FUNCTION ASSEMBLE_LWORD_FROM_WORDS (* this Function combines the 4 WORDS to a LWORD *)
  (* Standard: 61499-1; Description: Copyright (c) 2026 HR Agrartechnik GmbH This program and the accompanying materials are made available under the terms of the Eclipse Public License 2.0 which is available at https://www.eclipse.org/legal/epl-2.0/ SPDX-License-Identifier: EPL-2.0 *)
  (* Version 1.0, 2026-05-16, Franz Höpfinger, HR Agrartechnik, initial Implementation *)
  PACKAGE eclipse4diac::utils::assembling;
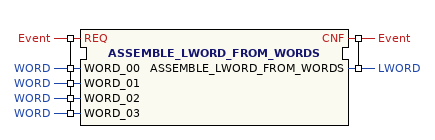
  EVENT_INPUT
    REQ WITH WORD_00, WORD_01, WORD_02, WORD_03;
  END_EVENT
  EVENT_OUTPUT
    CNF WITH ASSEMBLE_LWORD_FROM_WORDS;
  END_EVENT
  VAR_INPUT
    WORD_00 : WORD;
    WORD_01 : WORD;
    WORD_02 : WORD;
    WORD_03 : WORD;
  END_VAR
  VAR_OUTPUT
    ASSEMBLE_LWORD_FROM_WORDS : LWORD;
  END_VAR
  BODY IN ST:
PACKAGE eclipse4diac::utils::assembling;

(* this Function combines the 4 WORDS to a LWORD *)
FUNCTION ASSEMBLE_LWORD_FROM_WORDS : LWORD

VAR_INPUT
	WORD_00 : WORD;
	WORD_01 : WORD;
	WORD_02 : WORD;
	WORD_03 : WORD;
END_VAR

ASSEMBLE_LWORD_FROM_WORDS.%W0 := WORD_00;
ASSEMBLE_LWORD_FROM_WORDS.%W1 := WORD_01;
ASSEMBLE_LWORD_FROM_WORDS.%W2 := WORD_02;
ASSEMBLE_LWORD_FROM_WORDS.%W3 := WORD_03;

END_FUNCTION
  END_BODY
END_FUNCTION
